(* PLC project CoDeSys External Library Template, WAGO e!COCKPIT e!COCKPIT, author 3S - Smart Software Solutions GmbH *)
(* stored: creationDateTime 2019-10-29T12:22:40.6817378, version 3.5.5.30, modificationDateTime 2019-10-24T14:40:07.960949, organization 3S - Smart Software Solutions GmbH *)
(* Library project template with all possible element types, docu and a sample project structure *)

FUNCTION_BLOCK fbPPPSDestratyfikatorTBOX
  VAR_INPUT
    sKomunikat : alSTRINGKomunikat;  (* komunikat z systemu zewnętrznego *)
    intTablicaKomunikatowRozmiar : INT;  (* rozmiar tablicy danych wysyłkowych *)
    intModbusOdczytZapisZadanieRozmiar : INT;  (* rozmiar tablicy danych modbusa *)
    xTablicaKomunikatowHold : BOOL;  (* wstrzymanie komunikacji mniej ważnych komunikatów *)
    sIdInstancji : STRING;  (* parametr ID rolety np NS02L*202IBM**** *)
    sIdAplikacji : STRING;  (* parametr ID aplikacji np SO*******ECL*000 *)
    sMnemonik : STRING;  (* mnemonik właściciela - BCB* *)
    sMACAdres : STRING;  (* MAC adres sterownika *)
    sDaneZapasowe : STRING;  (* 6 znaków zapasu *)
    tCzasOpoznieniaRestartu : TIME;  (* czas opóźnienia po którym zaczynają być raportowane wartości *)
    tCzasOpoznieniaAlarmu : TIME := TIME#1m0s0ms;  (* czas opóźnienia po którym zaczynają być raportowane wartości *)
    bAdres : BYTE;
    tMinimalnyCzasRaportowania : TIME;
    tMaksymalnyCzasRaportowania : TIME;
    xAutonomizacja : BOOL;
    xAutonomizacjaSztuczna : BOOL;
  END_VAR
  VAR_IN_OUT
    arModbusOdczytCykliczny : ARRAY[1..5000] OF typModbusOdczytCykliczny;
    arModbusStatusKomunikacji : ARRAY[1..256] OF INT;
    arModbusOdczytZapisZadanie : ARRAY[1..1000] OF typModbusOdczytZapisZadanie;
    intModbusOdczytZapisZadanieZnacznikZapisu : INT;
    arTablicaKomunikatow : alARRAYTablicaKomunikatow;
    intTablicaKomunikatowZnacznikZapisu : INT;
  END_VAR
  VAR
    xPoInicjalizacji : BOOL := FALSE;  (* Inicjalizacja *)
    fbInicjalizacyjnyTimer : TON;
    tCzasInicjalizacji : TIME := TIME#30s0ms;
    xPierwszySkan : BOOL := TRUE;  (* Definicje zmiennych do odczytu wartości z modbusa *)
    intPetlaPierwszySkan : INT := 1;
    sDane : alSTRINGKomunikat;  (* Definicje do komunikacji z IZE *)
    sWyslanyKomunikat : alSTRINGKomunikat;
    sWyslanyKomunikatDummy : alSTRINGKomunikat;
    xZadanieRaportu : BOOL;
    sKomunikatPamiec : alSTRINGKomunikat;
    intPetla : INT;
    arErrorStan : ARRAY[0..10] OF INT;  (* tablica przechowująca statusy alarmowe *)
    arErrorKlasa : ARRAY[0..10] OF INT;  (* tablica przechowująca klasy danych alarmów *)
    xRaport : BOOL := FALSE;
    sTempWartoscAtrybutu : STRING;
    xOverFlow : BOOL;
    fbTimerBrakuKomunikacji : TON;  (* Kontrola komunikacji urządzenia *)
    xBrakKomunikacjiPLC : BOOL;
    xBrakKomunikacjiIZE : BOOL;
    intBlokadaWykonywaniaRozkazow : INT;  (* Parametry *)
    intBlokadaWykonywaniaRozkazowZaraportowana : INT;
    wSoftwareVersion : WORD;
    wTrybPracy : WORD;  (* 1 - wyłączony; 2 - auto (depend), 3 - auto (independ), 4 - manual *)
    rTrybPracy : REAL;
    rTrybPracyZaraportowana : REAL;
    wPredkoscWentylatora : WORD;  (* 0 - wyłączony; 1..33 - I bieg; 34..66 - drugi bieg; 67..100 - trzeci bieg *)
    rPredkoscWentylatora : REAL;
    rPredkoscWentylatoraZaraportowana : REAL;
    fbPredkoscWentylatora : fbFiltrWartoscAnalogowa;
    wTemperaturaReferencyjna : WORD;  (* 50..450 (10 = 1 st. C) *)
    rTemperaturaReferencyjna : REAL;
    rTemperaturaReferencyjnaZaraportowana : REAL;
    wTemperaturaRzeczywista : WORD;  (* -600..600 (10 = 1 st. C) *)
    rTemperaturaRzeczywista : REAL;
    rTemperaturaRzeczywistaZaraportowana : REAL;
    fbTemperaturaRzeczywista : fbFiltrWartoscAnalogowa;
    rTemperaturaRzeczywistaPamiec : REAL;
    xBrakZmianyTemperatury : BOOL;
    fbBrakZmianyTemperaturyTimer : TON;
    xBladBrakZmianyTemperatury : BOOL;
    wTemperaturaReferencyjnaTrybManualny : WORD;  (* 50..450 (10 = 1 st. C) *)
    rTemperaturaReferencyjnaTrybManualny : REAL;
    rTemperaturaReferencyjnaTrybManualnyZaraportowana : REAL;
  END_VAR

            (*			
Autor:					Jan Bartczak, 2019-01-10 
Prawa majątkowe: 		Solwena Sp. z o.o., 
Aktualizacje:			2019-01-28-AWy: Odczyt rejestrów temperatury ref., zadanej, prędkości wentylatora etc. Komunikacja z IZE.
						2019-02-06-AWy: Alarm braku komunikacji
						2019-05-16-AWy: Modyfikacja warunku na raportowanie. Dopisane: AND arModbusStatusKomunikacji[bAdres] = enumModbusStatus.KomunikacjaPrawidlowa AND xPoInicjalizacji 
						
Opis:					fb służy do komunikacji z zadajnikiem destratyfikatorów - T-BOX'em
				
*)


// Inicjalizacja sterownika
fbInicjalizacyjnyTimer(IN := (NOT xPoInicjalizacji AND arModbusStatusKomunikacji[bAdres] = enumModbusStatus.KomunikacjaPrawidlowa) , PT := tCzasOpoznieniaRestartu);
IF fbInicjalizacyjnyTimer.Q THEN
	rTrybPracyZaraportowana := rTrybPracy;
	rPredkoscWentylatoraZaraportowana := rPredkoscWentylatora;
	rTemperaturaReferencyjnaZaraportowana := rTemperaturaReferencyjna;
	rTemperaturaRzeczywistaZaraportowana := rTemperaturaRzeczywista;
	rTemperaturaReferencyjnaTrybManualnyZaraportowana := rTemperaturaReferencyjnaTrybManualny;
	xPoInicjalizacji := TRUE;
END_IF
//

IF xAutonomizacjaSztuczna = TRUE THEN
	xAutonomizacja := TRUE;
END_IF 

// Kontrola komunikacji
fbTimerBrakuKomunikacji(IN := arModbusStatusKomunikacji[bAdres] = enumModbusStatus.BrakKomunikacji, PT := T#60S);
IF fbTimerBrakuKomunikacji.Q THEN
	xBrakKomunikacjiPLC := TRUE;
ELSE
	xBrakKomunikacjiPLC := FALSE;
END_IF

IF xAutonomizacja THEN
	xBrakKomunikacjiIZE := TRUE;
ELSE
	xBrakKomunikacjiIZE := FALSE;
END_IF
//

IF xPierwszySkan THEN
	xPierwszySkan := FALSE;
	WHILE arModbusOdczytCykliczny[intPetlaPierwszySkan].bAdresUrzadzenia <> 0 DO
		intPetlaPierwszySkan := intPetlaPierwszySkan + 1;
	END_WHILE

	arModbusOdczytCykliczny[intPetlaPierwszySkan].bAdresUrzadzenia := bAdres;
	arModbusOdczytCykliczny[intPetlaPierwszySkan].bFunkcja := TO_BYTE(enumModbusKodyFunkcji.OdczytNRejestrowWejsciowych);
	arModbusOdczytCykliczny[intPetlaPierwszySkan].uiAdresRejestru := 3;
	arModbusOdczytCykliczny[intPetlaPierwszySkan].ltCzestotliwosc := TIME_TO_LTIME(tMinimalnyCzasRaportowania);
	arModbusOdczytCykliczny[intPetlaPierwszySkan].pZmiennaReferencyjna := ADR(wSoftwareVersion);
	intPetlaPierwszySkan := intPetlaPierwszySkan + 1;

	arModbusOdczytCykliczny[intPetlaPierwszySkan].bAdresUrzadzenia := bAdres;
	arModbusOdczytCykliczny[intPetlaPierwszySkan].bFunkcja := TO_BYTE(enumModbusKodyFunkcji.OdczytNRejestrowWejsciowych);
	arModbusOdczytCykliczny[intPetlaPierwszySkan].uiAdresRejestru := 5;
	arModbusOdczytCykliczny[intPetlaPierwszySkan].ltCzestotliwosc := TIME_TO_LTIME(tMinimalnyCzasRaportowania);
	arModbusOdczytCykliczny[intPetlaPierwszySkan].pZmiennaReferencyjna := ADR(wTemperaturaRzeczywista);
	intPetlaPierwszySkan := intPetlaPierwszySkan + 1;		

	arModbusOdczytCykliczny[intPetlaPierwszySkan].bAdresUrzadzenia := bAdres;
	arModbusOdczytCykliczny[intPetlaPierwszySkan].bFunkcja := TO_BYTE(enumModbusKodyFunkcji.OdczytNRejestrow);
	arModbusOdczytCykliczny[intPetlaPierwszySkan].uiAdresRejestru := 16#1004;
	arModbusOdczytCykliczny[intPetlaPierwszySkan].ltCzestotliwosc := TIME_TO_LTIME(tMinimalnyCzasRaportowania);
	arModbusOdczytCykliczny[intPetlaPierwszySkan].pZmiennaReferencyjna := ADR(wTrybPracy);
	intPetlaPierwszySkan := intPetlaPierwszySkan + 1;	
	
	arModbusOdczytCykliczny[intPetlaPierwszySkan].bAdresUrzadzenia := bAdres;
	arModbusOdczytCykliczny[intPetlaPierwszySkan].bFunkcja := TO_BYTE(enumModbusKodyFunkcji.OdczytNRejestrow);
	arModbusOdczytCykliczny[intPetlaPierwszySkan].uiAdresRejestru := 16#1005;
	arModbusOdczytCykliczny[intPetlaPierwszySkan].ltCzestotliwosc := TIME_TO_LTIME(tMinimalnyCzasRaportowania);
	arModbusOdczytCykliczny[intPetlaPierwszySkan].pZmiennaReferencyjna := ADR(wPredkoscWentylatora);
	intPetlaPierwszySkan := intPetlaPierwszySkan + 1;

	arModbusOdczytCykliczny[intPetlaPierwszySkan].bAdresUrzadzenia := bAdres;
	arModbusOdczytCykliczny[intPetlaPierwszySkan].bFunkcja := TO_BYTE(enumModbusKodyFunkcji.OdczytNRejestrow);
	arModbusOdczytCykliczny[intPetlaPierwszySkan].uiAdresRejestru := 16#1006;
	arModbusOdczytCykliczny[intPetlaPierwszySkan].ltCzestotliwosc := TIME_TO_LTIME(tMinimalnyCzasRaportowania);
	arModbusOdczytCykliczny[intPetlaPierwszySkan].pZmiennaReferencyjna := ADR(wTemperaturaReferencyjna);
	intPetlaPierwszySkan := intPetlaPierwszySkan + 1;		
	
	arModbusOdczytCykliczny[intPetlaPierwszySkan].bAdresUrzadzenia := bAdres;
	arModbusOdczytCykliczny[intPetlaPierwszySkan].bFunkcja := TO_BYTE(enumModbusKodyFunkcji.OdczytNRejestrow);
	arModbusOdczytCykliczny[intPetlaPierwszySkan].uiAdresRejestru := 16#1007;
	arModbusOdczytCykliczny[intPetlaPierwszySkan].ltCzestotliwosc := TIME_TO_LTIME(tMinimalnyCzasRaportowania);
	arModbusOdczytCykliczny[intPetlaPierwszySkan].pZmiennaReferencyjna := ADR(wTemperaturaReferencyjnaTrybManualny);
	intPetlaPierwszySkan := intPetlaPierwszySkan + 1;					
END_IF

// Przeliczenie zmiennych
rTrybPracy := WORD_TO_REAL(wTrybPracy);

fbPredkoscWentylatora(	rWartoscWejsciowa := WORD_TO_REAL(wPredkoscWentylatora),
						rDeadband := 5,
						tCzasMinimalny := tMinimalnyCzasRaportowania,
						tCzasMaksymalny := tMaksymalnyCzasRaportowania,
						rWynikMnoznik := 1,
						rWynikOffset := 0,
						rWartoscWejsciowaZaraportowana := rPredkoscWentylatoraZaraportowana,
						rWartoscWyjsciowa => rPredkoscWentylatora);
						
rTemperaturaReferencyjna := WORD_TO_REAL(wTemperaturaReferencyjna)*0.1 + 273.15;

fbTemperaturaRzeczywista(	rWartoscWejsciowa := WORD_TO_REAL(wTemperaturaRzeczywista),
							rDeadband := 0.5,
							tCzasMinimalny := tMinimalnyCzasRaportowania,
							tCzasMaksymalny := tMaksymalnyCzasRaportowania,
							rWynikMnoznik := 0.1,
							rWynikOffset := 273.15,
							rWartoscWejsciowaZaraportowana := rTemperaturaRzeczywistaZaraportowana,
							rWartoscWyjsciowa => rTemperaturaRzeczywista);
							
rTemperaturaReferencyjnaTrybManualny := WORD_TO_REAL(wTemperaturaReferencyjnaTrybManualny)*0.1 + 273.15;
//					
						
						
// Obsluga komunikatu przychodzacego z IZE
IF sKomunikat <> sKomunikatPamiec AND xPoInicjalizacji THEN
	sKomunikatPamiec := sKomunikat;
	IF fnIDOdbiorcyMatch(sKomunikat , sIdInstancji) THEN
		sDane := '';
		// Rozkaz typu C
		IF fnKomunikatTyp(sKomunikat) = 'C' AND NOT xAutonomizacja THEN
			IF fnKomunikatDaneSzukajWartosci(sKomunikat,'BLOK=') = '0' THEN
				IF intBlokadaWykonywaniaRozkazow = 1 THEN
					intBlokadaWykonywaniaRozkazow := 0;
					xRaport := TRUE;
					ELSE	
					IF sDane <> '' THEN
					sDane := CONCAT(sDane , ';');
					END_IF
					sDane := CONCAT(sDane , 'BLOK=0');
				END_IF
			END_IF
			IF fnKomunikatDaneSzukajWartosci(sKomunikat,'BLOK=') = '1' THEN
				IF intBlokadaWykonywaniaRozkazow = 0 THEN
					intBlokadaWykonywaniaRozkazow := 1;
					xRaport := TRUE;
					ELSE
					IF sDane <> '' THEN
					sDane := CONCAT(sDane , ';');
					END_IF					
					sDane := CONCAT(sDane , 'BLOK=1');
				END_IF
			END_IF
		END_IF
				
		// Zapytanie typu Q
		IF fnKomunikatTyp(sKomunikat) = 'Q' AND arModbusStatusKomunikacji[bAdres] = enumModbusStatus.KomunikacjaPrawidlowa THEN
			IF fnKomunikatDaneSzukajWartosci(sKomunikat , 'BLOK=') = '?' OR fnKomunikatDaneSzukajWartosci(sKomunikat , 'ALL=') = '?' THEN
				fnKomunikatDaneDodaj_xOverFlow(sDane := sDane , sAtrybut := 'BLOK=' , sWartosc := INT_TO_STRING(intBlokadaWykonywaniaRozkazow) , xOverFlow := xOverFlow);	
				IF xOverFlow = TRUE THEN
					fnZapiszKomunikat(	sCalyKomunikat := '' ,
								sTypKomunikatu := 'A' ,
								sMnemonik := sMnemonik ,
								sMACAdres := sMACAdres ,
								sIDNadawcy := sIdInstancji ,
								sIDOdbiorcy := sIdAplikacji ,
								sDaneZapasowe := sDaneZapasowe ,
								sDane := sDane ,
								arTablicaKomunikatow := arTablicaKomunikatow ,
								intTablicaKomunikatowZnacznikZapisu := intTablicaKomunikatowZnacznikZapisu ,
								intTablicaKomunikatowRozmiar := intTablicaKomunikatowRozmiar ,
								sWyslanyKomunikat := sWyslanyKomunikatDummy);
					sDane := '';
				END_IF
			END_IF
			IF fnKomunikatDaneSzukajWartosci(sKomunikat , 'TRYBPRACY=') = '?' OR fnKomunikatDaneSzukajWartosci(sKomunikat , 'ALL=') = '?' THEN
				fnKomunikatDaneDodaj_xOverFlow(sDane := sDane , sAtrybut := 'TRYBPRACY=' , sWartosc := REAL_TO_STRING(rTrybPracy) , xOverFlow := xOverFlow);	
				IF xOverFlow = TRUE THEN
					fnZapiszKomunikat(	sCalyKomunikat := '' ,
								sTypKomunikatu := 'A' ,
								sMnemonik := sMnemonik ,
								sMACAdres := sMACAdres ,
								sIDNadawcy := sIdInstancji ,
								sIDOdbiorcy := sIdAplikacji ,
								sDaneZapasowe := sDaneZapasowe ,
								sDane := sDane ,
								arTablicaKomunikatow := arTablicaKomunikatow ,
								intTablicaKomunikatowZnacznikZapisu := intTablicaKomunikatowZnacznikZapisu ,
								intTablicaKomunikatowRozmiar := intTablicaKomunikatowRozmiar ,
								sWyslanyKomunikat := sWyslanyKomunikatDummy);
					sDane := '';
				END_IF
			END_IF		
			IF fnKomunikatDaneSzukajWartosci(sKomunikat , 'PREDKOSCWENT=') = '?' OR fnKomunikatDaneSzukajWartosci(sKomunikat , 'ALL=') = '?' THEN
				fnKomunikatDaneDodaj_xOverFlow(sDane := sDane , sAtrybut := 'PREDKOSCWENT=' , sWartosc := REAL_TO_STRING(rPredkoscWentylatora) , xOverFlow := xOverFlow);	
				IF xOverFlow = TRUE THEN
					fnZapiszKomunikat(	sCalyKomunikat := '' ,
								sTypKomunikatu := 'A' ,
								sMnemonik := sMnemonik ,
								sMACAdres := sMACAdres ,
								sIDNadawcy := sIdInstancji ,
								sIDOdbiorcy := sIdAplikacji ,
								sDaneZapasowe := sDaneZapasowe ,
								sDane := sDane ,
								arTablicaKomunikatow := arTablicaKomunikatow ,
								intTablicaKomunikatowZnacznikZapisu := intTablicaKomunikatowZnacznikZapisu ,
								intTablicaKomunikatowRozmiar := intTablicaKomunikatowRozmiar ,
								sWyslanyKomunikat := sWyslanyKomunikatDummy);
					sDane := '';
				END_IF
			END_IF		
			IF fnKomunikatDaneSzukajWartosci(sKomunikat , 'TEMPREF=') = '?' OR fnKomunikatDaneSzukajWartosci(sKomunikat , 'ALL=') = '?' THEN
				fnKomunikatDaneDodaj_xOverFlow(sDane := sDane , sAtrybut := 'TEMPREF=' , sWartosc := REAL_TO_STRING(rTemperaturaReferencyjna) , xOverFlow := xOverFlow);	
				IF xOverFlow = TRUE THEN
					fnZapiszKomunikat(	sCalyKomunikat := '' ,
								sTypKomunikatu := 'A' ,
								sMnemonik := sMnemonik ,
								sMACAdres := sMACAdres ,
								sIDNadawcy := sIdInstancji ,
								sIDOdbiorcy := sIdAplikacji ,
								sDaneZapasowe := sDaneZapasowe ,
								sDane := sDane ,
								arTablicaKomunikatow := arTablicaKomunikatow ,
								intTablicaKomunikatowZnacznikZapisu := intTablicaKomunikatowZnacznikZapisu ,
								intTablicaKomunikatowRozmiar := intTablicaKomunikatowRozmiar ,
								sWyslanyKomunikat := sWyslanyKomunikatDummy);
					sDane := '';
				END_IF
			END_IF		
			IF fnKomunikatDaneSzukajWartosci(sKomunikat , 'TEMPRZECZ=') = '?' OR fnKomunikatDaneSzukajWartosci(sKomunikat , 'ALL=') = '?' THEN
				fnKomunikatDaneDodaj_xOverFlow(sDane := sDane , sAtrybut := 'TEMPRZECZ=' , sWartosc := REAL_TO_STRING(rTemperaturaRzeczywista) , xOverFlow := xOverFlow);	
				IF xOverFlow = TRUE THEN
					fnZapiszKomunikat(	sCalyKomunikat := '' ,
								sTypKomunikatu := 'A' ,
								sMnemonik := sMnemonik ,
								sMACAdres := sMACAdres ,
								sIDNadawcy := sIdInstancji ,
								sIDOdbiorcy := sIdAplikacji ,
								sDaneZapasowe := sDaneZapasowe ,
								sDane := sDane ,
								arTablicaKomunikatow := arTablicaKomunikatow ,
								intTablicaKomunikatowZnacznikZapisu := intTablicaKomunikatowZnacznikZapisu ,
								intTablicaKomunikatowRozmiar := intTablicaKomunikatowRozmiar ,
								sWyslanyKomunikat := sWyslanyKomunikatDummy);
					sDane := '';
				END_IF
			END_IF		
			IF fnKomunikatDaneSzukajWartosci(sKomunikat , 'TEMPREFTRYBMAN=') = '?' OR fnKomunikatDaneSzukajWartosci(sKomunikat , 'ALL=') = '?' THEN
				fnKomunikatDaneDodaj_xOverFlow(sDane := sDane , sAtrybut := 'TEMPREFTRYBMAN=' , sWartosc := REAL_TO_STRING(rTemperaturaReferencyjnaTrybManualny) , xOverFlow := xOverFlow);	
				IF xOverFlow = TRUE THEN
					fnZapiszKomunikat(	sCalyKomunikat := '' ,
								sTypKomunikatu := 'A' ,
								sMnemonik := sMnemonik ,
								sMACAdres := sMACAdres ,
								sIDNadawcy := sIdInstancji ,
								sIDOdbiorcy := sIdAplikacji ,
								sDaneZapasowe := sDaneZapasowe ,
								sDane := sDane ,
								arTablicaKomunikatow := arTablicaKomunikatow ,
								intTablicaKomunikatowZnacznikZapisu := intTablicaKomunikatowZnacznikZapisu ,
								intTablicaKomunikatowRozmiar := intTablicaKomunikatowRozmiar ,
								sWyslanyKomunikat := sWyslanyKomunikatDummy);
					sDane := '';
				END_IF
			END_IF		
			// Pytanie o stany alarmów
			IF fnKomunikatDaneSzukajWartosci(sKomunikat , 'ALARM=') = '?' OR fnKomunikatDaneSzukajWartosci(sKomunikat , 'ALL=') = '?' THEN
				FOR intPetla := 1 TO 10 BY 1 DO
					// Raportowanie typu E (stanów alarmów) na zapytanie typu Q
					IF arErrorStan[intPetla] <> enumAlarmWartosc.StanNieznany THEN
						fnZapiszKomunikat(	sCalyKomunikat := '' ,
											sTypKomunikatu := 'E' ,
											sMnemonik := sMnemonik ,
											sMACAdres := sMACAdres ,
											sIDNadawcy := sIdInstancji ,
											sIDOdbiorcy := sIdAplikacji ,
											sDaneZapasowe := sDaneZapasowe ,
											sDane := fnKomunikatDaneErrorRetry(xAktywny := arErrorStan[intPetla] = enumAlarmWartosc.StanAlarmowy , intKlasa := arErrorKlasa[intPetla] , intNumer := intPetla),
											arTablicaKomunikatow := arTablicaKomunikatow ,
											intTablicaKomunikatowZnacznikZapisu := intTablicaKomunikatowZnacznikZapisu ,
											intTablicaKomunikatowRozmiar := intTablicaKomunikatowRozmiar ,
											sWyslanyKomunikat := sWyslanyKomunikatDummy);
					END_IF
				END_FOR
			END_IF
		END_IF		
		// Raportowanie typu A na zapytanie Q
		IF sDane <> '' THEN
			fnZapiszKomunikat(	sCalyKomunikat := '' ,
								sTypKomunikatu := 'A' ,
								sMnemonik := sMnemonik ,
								sMACAdres := sMACAdres ,
								sIDNadawcy := sIdInstancji ,
								sIDOdbiorcy := sIdAplikacji ,
								sDaneZapasowe := sDaneZapasowe ,
								sDane := sDane ,
								arTablicaKomunikatow := arTablicaKomunikatow ,
								intTablicaKomunikatowZnacznikZapisu := intTablicaKomunikatowZnacznikZapisu ,
								intTablicaKomunikatowRozmiar := intTablicaKomunikatowRozmiar ,
								sWyslanyKomunikat := sWyslanyKomunikatDummy);
		END_IF
	END_IF
END_IF

// Raportowanie typu M do IZE wartosci odczytanych z Modbusa	
IF 	(intBlokadaWykonywaniaRozkazow <> intBlokadaWykonywaniaRozkazowZaraportowana OR rTrybPracy <> rTrybPracyZaraportowana OR rPredkoscWentylatora <> rPredkoscWentylatoraZaraportowana OR
	rTemperaturaReferencyjna <> rTemperaturaReferencyjnaZaraportowana OR rTemperaturaRzeczywista <> rTemperaturaRzeczywistaZaraportowana OR 
	rTemperaturaReferencyjnaTrybManualny <> rTemperaturaReferencyjnaTrybManualnyZaraportowana)AND arModbusStatusKomunikacji[bAdres] = enumModbusStatus.KomunikacjaPrawidlowa AND xPoInicjalizacji THEN
	xRaport := TRUE;
END_IF

IF xRaport THEN
	sDane := '';
	xRaport := FALSE;
	IF intBlokadaWykonywaniaRozkazow <> intBlokadaWykonywaniaRozkazowZaraportowana THEN 
		intBlokadaWykonywaniaRozkazowZaraportowana := intBlokadaWykonywaniaRozkazow;
		fnKomunikatDaneDodaj_xOverFlow(sDane := sDane , sAtrybut := 'BLOK=' , sWartosc := INT_TO_STRING(intBlokadaWykonywaniaRozkazow) , xOverFlow := xOverFlow);	
	END_IF	
	IF xOverFlow = TRUE THEN
		fnZapiszKomunikat(	sCalyKomunikat := '' ,
					sTypKomunikatu := 'M' ,
					sMnemonik := sMnemonik ,
					sMACAdres := sMACAdres ,
					sIDNadawcy := sIdInstancji ,
					sIDOdbiorcy := sIdAplikacji ,
					sDaneZapasowe := sDaneZapasowe ,
					sDane := sDane ,
					arTablicaKomunikatow := arTablicaKomunikatow ,
					intTablicaKomunikatowZnacznikZapisu := intTablicaKomunikatowZnacznikZapisu ,
					intTablicaKomunikatowRozmiar := intTablicaKomunikatowRozmiar ,
					sWyslanyKomunikat := sWyslanyKomunikatDummy);
		sDane := '';
	END_IF
	// Tryb pracy
	IF rTrybPracy <> rTrybPracyZaraportowana THEN
		rTrybPracyZaraportowana := rTrybPracy;
		fnKomunikatDaneDodaj_xOverFlow(sDane := sDane , sAtrybut := 'TRYBPRACY=' , sWartosc := REAL_TO_STRING(rTrybPracy) , xOverFlow := xOverFlow);	
		IF xOverFlow = TRUE THEN
			fnZapiszKomunikat(	sCalyKomunikat := '' ,
						sTypKomunikatu := 'M' ,
						sMnemonik := sMnemonik ,
						sMACAdres := sMACAdres ,
						sIDNadawcy := sIdInstancji ,
						sIDOdbiorcy := sIdAplikacji ,
						sDaneZapasowe := sDaneZapasowe ,
						sDane := sDane ,
						arTablicaKomunikatow := arTablicaKomunikatow ,
						intTablicaKomunikatowZnacznikZapisu := intTablicaKomunikatowZnacznikZapisu ,
						intTablicaKomunikatowRozmiar := intTablicaKomunikatowRozmiar ,
						sWyslanyKomunikat := sWyslanyKomunikatDummy);
			sDane := '';
		END_IF	
	END_IF
	// Prędkość wentylatora
	IF rPredkoscWentylatora <> rPredkoscWentylatoraZaraportowana THEN
		rPredkoscWentylatoraZaraportowana := rPredkoscWentylatora;
		fnKomunikatDaneDodaj_xOverFlow(sDane := sDane , sAtrybut := 'PREDKOSCWENT=' , sWartosc := REAL_TO_STRING(rPredkoscWentylatora) , xOverFlow := xOverFlow);	
		IF xOverFlow = TRUE THEN
			fnZapiszKomunikat(	sCalyKomunikat := '' ,
						sTypKomunikatu := 'M' ,
						sMnemonik := sMnemonik ,
						sMACAdres := sMACAdres ,
						sIDNadawcy := sIdInstancji ,
						sIDOdbiorcy := sIdAplikacji ,
						sDaneZapasowe := sDaneZapasowe ,
						sDane := sDane ,
						arTablicaKomunikatow := arTablicaKomunikatow ,
						intTablicaKomunikatowZnacznikZapisu := intTablicaKomunikatowZnacznikZapisu ,
						intTablicaKomunikatowRozmiar := intTablicaKomunikatowRozmiar ,
						sWyslanyKomunikat := sWyslanyKomunikatDummy);
			sDane := '';
		END_IF	
	END_IF
	// Temperatura referencyjna
	IF rTemperaturaReferencyjna <> rTemperaturaReferencyjnaZaraportowana THEN
		rTemperaturaReferencyjnaZaraportowana := rTemperaturaReferencyjna;
		fnKomunikatDaneDodaj_xOverFlow(sDane := sDane , sAtrybut := 'TEMPREF=' , sWartosc := REAL_TO_STRING(rTemperaturaReferencyjna) , xOverFlow := xOverFlow);	
		IF xOverFlow = TRUE THEN
			fnZapiszKomunikat(	sCalyKomunikat := '' ,
						sTypKomunikatu := 'M' ,
						sMnemonik := sMnemonik ,
						sMACAdres := sMACAdres ,
						sIDNadawcy := sIdInstancji ,
						sIDOdbiorcy := sIdAplikacji ,
						sDaneZapasowe := sDaneZapasowe ,
						sDane := sDane ,
						arTablicaKomunikatow := arTablicaKomunikatow ,
						intTablicaKomunikatowZnacznikZapisu := intTablicaKomunikatowZnacznikZapisu ,
						intTablicaKomunikatowRozmiar := intTablicaKomunikatowRozmiar ,
						sWyslanyKomunikat := sWyslanyKomunikatDummy);
			sDane := '';
		END_IF	
	END_IF
	// Temperatura rzeczywista
	IF rTemperaturaRzeczywista <> rTemperaturaRzeczywistaZaraportowana THEN
		rTemperaturaRzeczywistaZaraportowana := rTemperaturaRzeczywista;
		fnKomunikatDaneDodaj_xOverFlow(sDane := sDane , sAtrybut := 'TEMPRZECZ=' , sWartosc := REAL_TO_STRING(rTemperaturaRzeczywista) , xOverFlow := xOverFlow);	
		IF xOverFlow = TRUE THEN
			fnZapiszKomunikat(	sCalyKomunikat := '' ,
						sTypKomunikatu := 'M' ,
						sMnemonik := sMnemonik ,
						sMACAdres := sMACAdres ,
						sIDNadawcy := sIdInstancji ,
						sIDOdbiorcy := sIdAplikacji ,
						sDaneZapasowe := sDaneZapasowe ,
						sDane := sDane ,
						arTablicaKomunikatow := arTablicaKomunikatow ,
						intTablicaKomunikatowZnacznikZapisu := intTablicaKomunikatowZnacznikZapisu ,
						intTablicaKomunikatowRozmiar := intTablicaKomunikatowRozmiar ,
						sWyslanyKomunikat := sWyslanyKomunikatDummy);
			sDane := '';
		END_IF	
	END_IF
	// Temperatura referencyjna trybu manulnego
	IF rTemperaturaReferencyjnaTrybManualny <> rTemperaturaReferencyjnaTrybManualnyZaraportowana THEN
		rTemperaturaReferencyjnaTrybManualnyZaraportowana := rTemperaturaReferencyjnaTrybManualny;
		fnKomunikatDaneDodaj_xOverFlow(sDane := sDane , sAtrybut := 'TEMPREFTRYBMAN=' , sWartosc := REAL_TO_STRING(rTemperaturaReferencyjnaTrybManualny) , xOverFlow := xOverFlow);	
		IF xOverFlow = TRUE THEN
			fnZapiszKomunikat(	sCalyKomunikat := '' ,
						sTypKomunikatu := 'M' ,
						sMnemonik := sMnemonik ,
						sMACAdres := sMACAdres ,
						sIDNadawcy := sIdInstancji ,
						sIDOdbiorcy := sIdAplikacji ,
						sDaneZapasowe := sDaneZapasowe ,
						sDane := sDane ,
						arTablicaKomunikatow := arTablicaKomunikatow ,
						intTablicaKomunikatowZnacznikZapisu := intTablicaKomunikatowZnacznikZapisu ,
						intTablicaKomunikatowRozmiar := intTablicaKomunikatowRozmiar ,
						sWyslanyKomunikat := sWyslanyKomunikatDummy);
			sDane := '';
		END_IF	
	END_IF
	IF sDane <> '' AND xPoInicjalizacji THEN
	fnZapiszKomunikat(	sCalyKomunikat := '' ,
						sTypKomunikatu := 'M' ,
						sMnemonik := sMnemonik ,
						sMACAdres := sMACAdres ,
						sIDNadawcy := sIdInstancji ,
						sIDOdbiorcy := sIdAplikacji ,
						sDaneZapasowe := sDaneZapasowe ,
						sDane := sDane ,
						arTablicaKomunikatow := arTablicaKomunikatow ,
						intTablicaKomunikatowZnacznikZapisu := intTablicaKomunikatowZnacznikZapisu ,
						intTablicaKomunikatowRozmiar := intTablicaKomunikatowRozmiar ,
						sWyslanyKomunikat := sWyslanyKomunikat);
	END_IF
END_IF

// Sprawdzanie czy pomiar temperatury działa (odczyt jest niepoprawny, jeśli nie zmienił wartości w przeciągu doby)
IF rTemperaturaRzeczywistaPamiec = rTemperaturaRzeczywista THEN
	xBrakZmianyTemperatury := TRUE;
ELSE
	xBrakZmianyTemperatury := FALSE;	
END_IF
fbBrakZmianyTemperaturyTimer(IN := xBrakZmianyTemperatury, PT := T#12H);
rTemperaturaRzeczywistaPamiec := rTemperaturaRzeczywista;
IF fbBrakZmianyTemperaturyTimer.Q THEN
	xBladBrakZmianyTemperatury := TRUE;
ELSE
	xBladBrakZmianyTemperatury := FALSE;
END_IF

// Alarm braku komunikacji MODBUS 
IF arErrorStan[enumPPPSDestratyfikatorTBOXError.BrakKomunikacji] <> enumAlarmWartosc.StanAlarmowy AND arModbusStatusKomunikacji[bAdres] = enumModbusStatus.BrakKomunikacji THEN
	arErrorStan[enumPPPSDestratyfikatorTBOXError.BrakKomunikacji] := enumAlarmWartosc.StanAlarmowy;
	arErrorKlasa[enumPPPSDestratyfikatorTBOXError.BrakKomunikacji] := enumPPPSDestratyfikatorTBOXErrorKlasa.BrakKomunikacji;
	IF xPoInicjalizacji THEN
		fnZapiszKomunikat(	sCalyKomunikat := '' ,
							sTypKomunikatu := 'E' ,
							sMnemonik := sMnemonik ,
							sMACAdres := sMACAdres ,
							sIDNadawcy := sIdInstancji ,
							sIDOdbiorcy := sIdAplikacji ,
							sDaneZapasowe := sDaneZapasowe ,
							sDane := fnKomunikatDaneError(xAktywny := TRUE , intKlasa := enumPPPSDestratyfikatorTBOXErrorKlasa.BrakKomunikacji , intNumer := enumPPPSDestratyfikatorTBOXError.BrakKomunikacji),
							arTablicaKomunikatow := arTablicaKomunikatow ,
							intTablicaKomunikatowZnacznikZapisu := intTablicaKomunikatowZnacznikZapisu ,
							intTablicaKomunikatowRozmiar := intTablicaKomunikatowRozmiar ,
							sWyslanyKomunikat := sWyslanyKomunikatDummy);
	END_IF
END_IF
IF arErrorStan[enumPPPSDestratyfikatorTBOXError.BrakKomunikacji] <> enumAlarmWartosc.StanNormalny AND arModbusStatusKomunikacji[bAdres] = enumModbusStatus.KomunikacjaPrawidlowa THEN
	arErrorStan[enumPPPSDestratyfikatorTBOXError.BrakKomunikacji] := enumAlarmWartosc.StanNormalny;
	arErrorKlasa[enumPPPSDestratyfikatorTBOXError.BrakKomunikacji] := enumPPPSDestratyfikatorTBOXErrorKlasa.BrakKomunikacji;
	IF xPoInicjalizacji THEN
		fnZapiszKomunikat(	sCalyKomunikat := '' ,
							sTypKomunikatu := 'E' ,
							sMnemonik := sMnemonik ,
							sMACAdres := sMACAdres ,
							sIDNadawcy := sIdInstancji ,
							sIDOdbiorcy := sIdAplikacji ,
							sDaneZapasowe := sDaneZapasowe ,
							sDane := fnKomunikatDaneError(xAktywny := FALSE , intKlasa := enumPPPSDestratyfikatorTBOXErrorKlasa.BrakKomunikacji , intNumer := enumPPPSDestratyfikatorTBOXError.BrakKomunikacji),
							arTablicaKomunikatow := arTablicaKomunikatow ,
							intTablicaKomunikatowZnacznikZapisu := intTablicaKomunikatowZnacznikZapisu ,
							intTablicaKomunikatowRozmiar := intTablicaKomunikatowRozmiar ,
							sWyslanyKomunikat := sWyslanyKomunikatDummy);
	END_IF
END_IF

// Alarm czujnika temperatury
IF arErrorStan[enumPPPSDestratyfikatorTBOXError.AlarmCzujnika] <> enumAlarmWartosc.StanAlarmowy AND xBladBrakZmianyTemperatury AND arModbusStatusKomunikacji[bAdres] = enumModbusStatus.KomunikacjaPrawidlowa THEN
	arErrorStan[enumPPPSDestratyfikatorTBOXError.AlarmCzujnika] := enumAlarmWartosc.StanAlarmowy;
	arErrorKlasa[enumPPPSDestratyfikatorTBOXError.AlarmCzujnika] := enumPPPSDestratyfikatorTBOXErrorKlasa.AlarmCzujnika;
	IF xPoInicjalizacji THEN
		fnZapiszKomunikat(	sCalyKomunikat := '' ,
							sTypKomunikatu := 'E' ,
							sMnemonik := sMnemonik ,
							sMACAdres := sMACAdres ,
							sIDNadawcy := sIdInstancji ,
							sIDOdbiorcy := sIdAplikacji ,
							sDaneZapasowe := sDaneZapasowe ,
							sDane := fnKomunikatDaneError(xAktywny := TRUE , intKlasa := enumPPPSDestratyfikatorTBOXErrorKlasa.AlarmCzujnika , intNumer := enumPPPSDestratyfikatorTBOXError.AlarmCzujnika),
							arTablicaKomunikatow := arTablicaKomunikatow ,
							intTablicaKomunikatowZnacznikZapisu := intTablicaKomunikatowZnacznikZapisu ,
							intTablicaKomunikatowRozmiar := intTablicaKomunikatowRozmiar ,
							sWyslanyKomunikat := sWyslanyKomunikatDummy);
	END_IF
END_IF
IF arErrorStan[enumPPPSDestratyfikatorTBOXError.AlarmCzujnika] <> enumAlarmWartosc.StanNormalny AND NOT xBladBrakZmianyTemperatury AND arModbusStatusKomunikacji[bAdres] = enumModbusStatus.KomunikacjaPrawidlowa THEN
	arErrorStan[enumPPPSDestratyfikatorTBOXError.AlarmCzujnika] := enumAlarmWartosc.StanNormalny;
	arErrorKlasa[enumPPPSDestratyfikatorTBOXError.AlarmCzujnika] := enumPPPSDestratyfikatorTBOXErrorKlasa.AlarmCzujnika;
	IF xPoInicjalizacji THEN
		fnZapiszKomunikat(	sCalyKomunikat := '' ,
							sTypKomunikatu := 'E' ,
							sMnemonik := sMnemonik ,
							sMACAdres := sMACAdres ,
							sIDNadawcy := sIdInstancji ,
							sIDOdbiorcy := sIdAplikacji ,
							sDaneZapasowe := sDaneZapasowe ,
							sDane := fnKomunikatDaneError(xAktywny := FALSE , intKlasa := enumPPPSDestratyfikatorTBOXErrorKlasa.AlarmCzujnika , intNumer := enumPPPSDestratyfikatorTBOXError.AlarmCzujnika),
							arTablicaKomunikatow := arTablicaKomunikatow ,
							intTablicaKomunikatowZnacznikZapisu := intTablicaKomunikatowZnacznikZapisu ,
							intTablicaKomunikatowRozmiar := intTablicaKomunikatowRozmiar ,
							sWyslanyKomunikat := sWyslanyKomunikatDummy);
	END_IF
END_IF

          
END_FUNCTION_BLOCK
